// Mitsubishi GX Works2 project: LocalPlc   PLC: Q03UDE

PROGRAM ROBOT
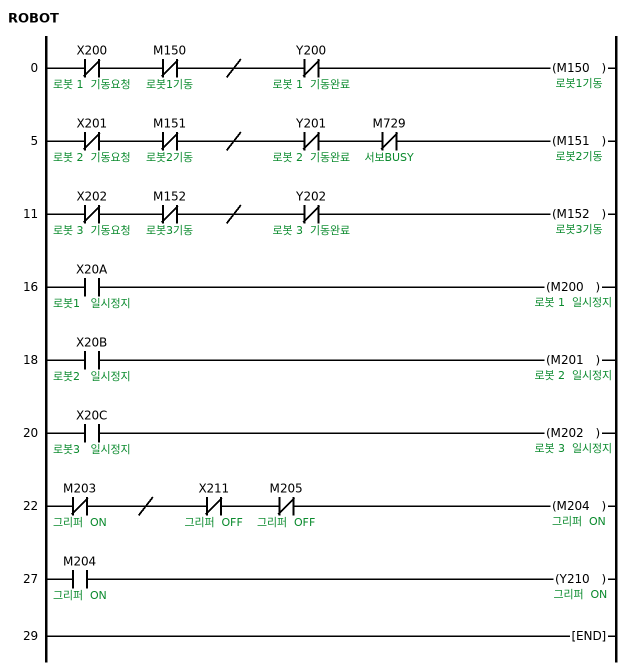
0     LDI     X200  ; 로봇 1  기동요청
      ANI     M150  ; 로봇1기동
      INV
      ANI     Y200  ; 로봇 1  기동완료
      OUT     M150  ; 로봇1기동
5     LDI     X201  ; 로봇 2  기동요청
      ANI     M151  ; 로봇2기동
      INV
      ANI     Y201  ; 로봇 2  기동완료
      ANI     M729  ; 서보BUSY
      OUT     M151  ; 로봇2기동
11    LDI     X202  ; 로봇 3  기동요청
      ANI     M152  ; 로봇3기동
      INV
      ANI     Y202  ; 로봇 3  기동완료
      OUT     M152  ; 로봇3기동
16    LD      X20A  ; 로봇1   일시정지
      OUT     M200  ; 로봇 1  일시정지
18    LD      X20B  ; 로봇2   일시정지
      OUT     M201  ; 로봇 2  일시정지
20    LD      X20C  ; 로봇3   일시정지
      OUT     M202  ; 로봇 3  일시정지
22    LDI     M203  ; 그리퍼  ON
      INV
      ANI     X211  ; 그리퍼  OFF
      ANI     M205  ; 그리퍼  OFF
      OUT     M204  ; 그리퍼  ON
27    LD      M204  ; 그리퍼  ON
      OUT     Y210  ; 그리퍼  ON
29    END
END_PROGRAM

PROGRAM HMI_BT
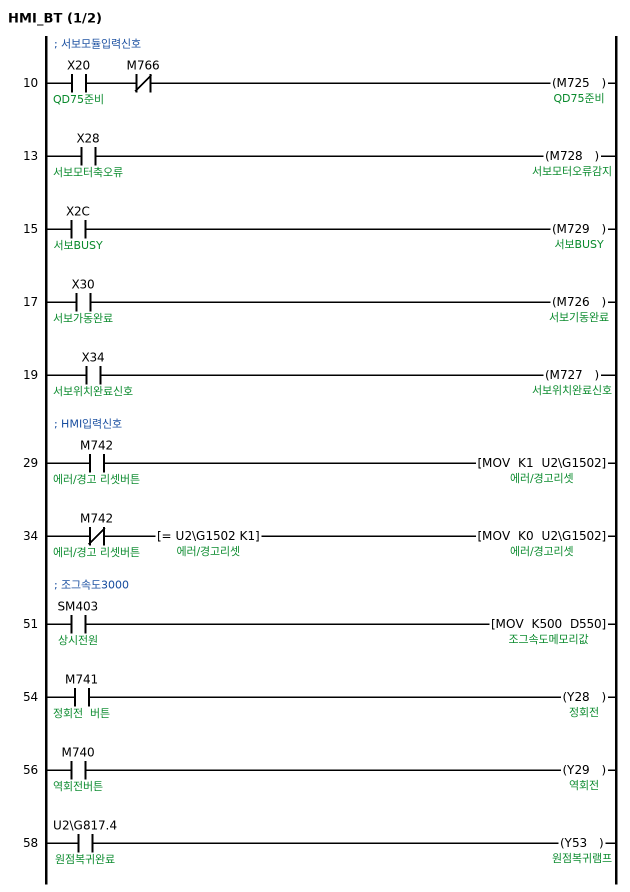
; 서보모듈입력신호
10    LD      X20  ; QD75준비
      ANI     M766
      OUT     M725  ; QD75준비
13    LD      X28  ; 서보모터축오류
      OUT     M728  ; 서보모터오류감지
15    LD      X2C  ; 서보BUSY
      OUT     M729  ; 서보BUSY
17    LD      X30  ; 서보가동완료
      OUT     M726  ; 서보기동완료
19    LD      X34  ; 서보위치완료신호
      OUT     M727  ; 서보위치완료신호
; HMI입력신호
29    LD      M742  ; 에러/경고 리셋버튼
      MOV     K1 U2\G1502  ; 에러/경고리셋
34    LDI     M742  ; 에러/경고 리셋버튼
      AND=    U2\G1502 K1  ; 에러/경고리셋
      MOV     K0 U2\G1502
; 조그속도3000
51    LD      SM403  ; 상시전원
      MOV     K500 D550  ; 조그속도메모리값
54    LD      M741  ; 정회전  버튼
      OUT     Y28  ; 정회전
56    LD      M740  ; 역회전버튼
      OUT     Y29  ; 역회전
58    LD      U2\G817.4  ; 원점복귀완료
      OUT     Y53  ; 원점복귀램프
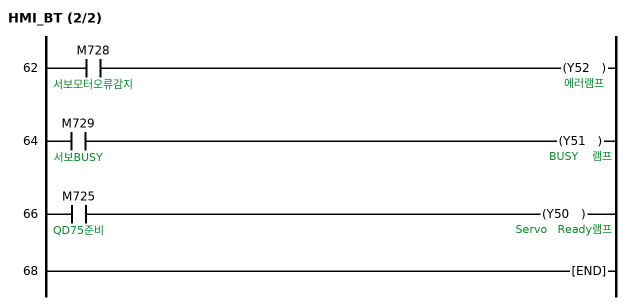
62    LD      M728  ; 서보모터오류감지
      OUT     Y52  ; 에러램프
64    LD      M729  ; 서보BUSY
      OUT     Y51  ; BUSY    램프
66    LD      M725  ; QD75준비
      OUT     Y50  ; Servo   Ready램프
68    END
END_PROGRAM

PROGRAM HMI_D
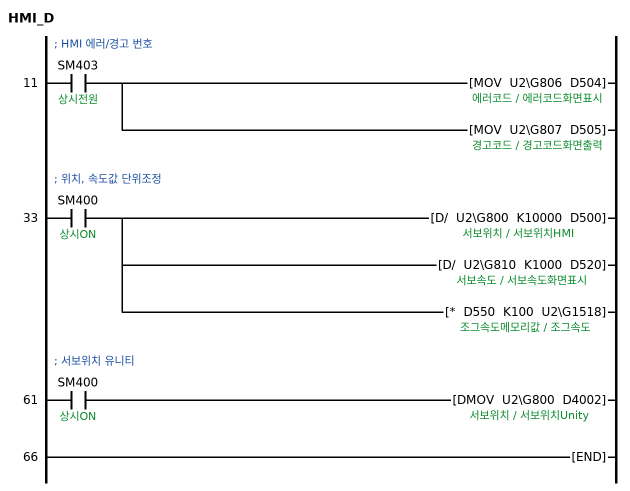
; HMI 에러/경고 번호
11    LD      SM403  ; 상시전원
      MOV     U2\G806 D504  ; 에러코드 / 에러코드화면표시
      MOV     U2\G807 D505  ; 경고코드 / 경고코드화면출력
; 위치, 속도값 단위조정
33    LD      SM400  ; 상시ON
      D/      U2\G800 K10000 D500  ; 서보위치 / 서보위치HMI
      D/      U2\G810 K1000 D520  ; 서보속도 / 서보속도화면표시
      *       D550 K100 U2\G1518  ; 조그속도메모리값 / 조그속도
; 서보위치 유니티
61    LD      SM400  ; 상시ON
      DMOV    U2\G800 D4002  ; 서보위치Unity
66    END
END_PROGRAM

PROGRAM SV_SEQUE
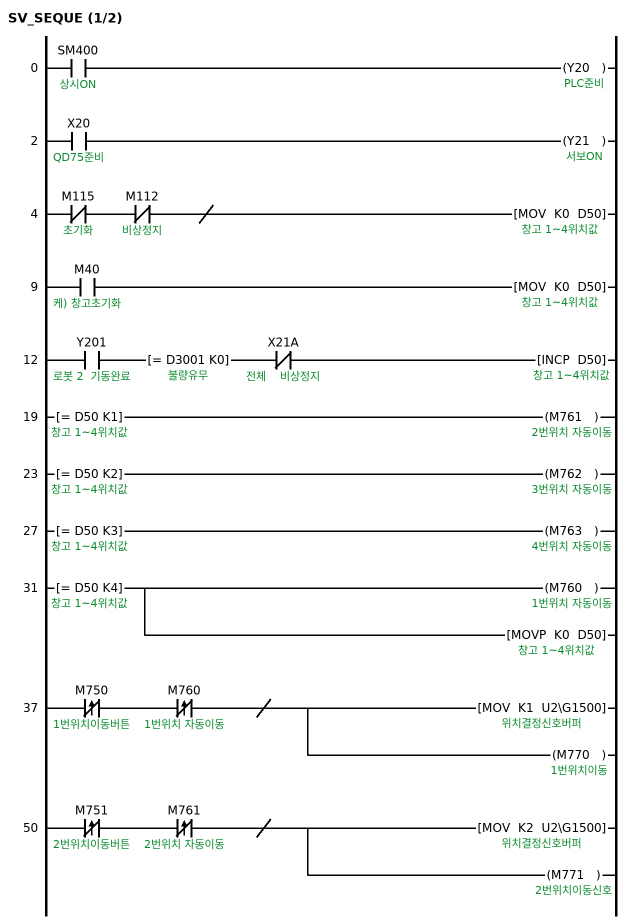
0     LD      SM400  ; 상시ON
      OUT     Y20  ; PLC준비
2     LD      X20  ; QD75준비
      OUT     Y21  ; 서보ON
4     LDI     M115  ; 초기화
      ANI     M112  ; 비상정지
      INV
      MOV     K0 D50  ; 창고 1~4위치값
9     LD      M40  ; 케) 창고초기화
      MOV     K0 D50
12    LD      Y201  ; 로봇 2  기동완료
      AND=    D3001 K0  ; 불량유무
      ANI     X21A  ; 전체    비상정지
      INCP    D50
19    LD=     D50 K1  ; 창고 1~4위치값
      OUT     M761  ; 2번위치 자동이동
23    LD=     D50 K2  ; 창고 1~4위치값
      OUT     M762  ; 3번위치 자동이동
27    LD=     D50 K3  ; 창고 1~4위치값
      OUT     M763  ; 4번위치 자동이동
31    LD=     D50 K4  ; 창고 1~4위치값
      OUT     M760  ; 1번위치 자동이동
      MOVP    K0 D50
37    LDPI    M750  ; 1번위치이동버튼
      ANDPI   M760  ; 1번위치 자동이동
      INV
      MOV     K1 U2\G1500  ; 위치결정신호버퍼
      OUT     M770  ; 1번위치이동
50    LDPI    M751  ; 2번위치이동버튼
      ANDPI   M761  ; 2번위치 자동이동
      INV
      MOV     K2 U2\G1500
      OUT     M771  ; 2번위치이동신호
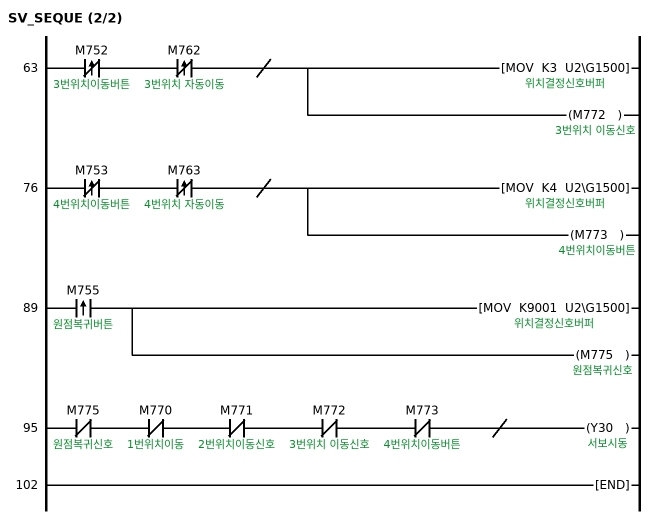
63    LDPI    M752  ; 3번위치이동버튼
      ANDPI   M762  ; 3번위치 자동이동
      INV
      MOV     K3 U2\G1500
      OUT     M772  ; 3번위치 이동신호
76    LDPI    M753  ; 4번위치이동버튼
      ANDPI   M763  ; 4번위치 자동이동
      INV
      MOV     K4 U2\G1500
      OUT     M773  ; 4번위치이동버튼
89    LDP     M755  ; 원점복귀버튼
      MOV     K9001 U2\G1500
      OUT     M775  ; 원점복귀신호
95    LDI     M775  ; 원점복귀신호
      ANI     M770  ; 1번위치이동
      ANI     M771  ; 2번위치이동신호
      ANI     M772  ; 3번위치 이동신호
      ANI     M773  ; 4번위치이동버튼
      INV
      OUT     Y30  ; 서보시동
102   END
END_PROGRAM

// device comments not shown above
X217  ; 로봇1   원점복귀
X218  ; 로봇2   원점복귀
X219  ; 로봇3   원점복귀
M50  ; 2번로봇완료신호
M51  ; 창고다음위치
M100  ; 완료저장->M101
M101  ; 로봇 2  기동
M102  ; 로봇 3  기동
M110  ; 자동시작
M111  ; 일시정지
M114  ; 자동운전
M210  ; 원점복귀입력
M215  ; 원점복귀이동신호
M300  ; 역회전   조작
M315  ; 원점복귀이동입력
M350  ; 1번위치
M351  ; 2번위치
M352  ; 3번위치
M500  ; HMI속도입력버튼
M555  ; 위치값입력버튼
M565  ; 원하는위치이동
M566  ; 래더짜세요
M700  ; 현위치값 임시저장
M701  ; 저장위치이동
M720  ; 위치임시저장삭제
M721  ; 2번위치이동버튼
M722  ; 3번위치이동버튼
M730  ; 조그속도3000버튼
M754  ; 원점기동신호2
M776  ; 원점복귀신호표시
M780  ; 원점기동자기유지
D0  ; 컨트롤 데이터
D2  ; 기동번호
D300  ; 서보스텝
D501  ; 서보위치현재값
D502  ; 서보속도값이동
D503  ; 현위치->임시저장
D560  ; HMI표시된위치값
D1000  ; 위치입력
D1500  ; 서보속도화면표시
D2000  ; HMI속도입력
D3050  ; 조그속도메모리값
D3060  ; HMI표시된위치값
D4000  ; 속도입력
T0  ; 역회전속도딜레이
